FUNCTION FC_CycleTimeToString : STRING(20);
VAR_INPUT
	CycleTime	: DWORD;
END_VAR
VAR
    TempStr : STRING(20);
    Thousands : UDINT;
    Remainder : UDINT;
	sRemainder : STRING(3);
END_VAR

(* Calcolo delle migliaia e del resto *)
Thousands := CycleTime / 1000;
Remainder := CycleTime MOD 1000;

(* Creazione della stringa con il formato richiesto *)
IF Thousands = 0 THEN
    // Se < 1000: stampiamo il valore diretto
	TempStr := '0.';
    TempStr := CONCAT(TempStr, DWORD_TO_STRING(CycleTime));
ELSE
     // Se >= 1000: separiamo migliaia e resto, es. 10901 -> "10.901"
    TempStr := UDINT_TO_STRING(Thousands);

    // Converto il resto in stringa
    sRemainder := UDINT_TO_STRING(Remainder);

    // Aggiungo eventuali zeri a sinistra, per avere sempre 3 cifre nel resto
    IF LEN(sRemainder) = 1 THEN
        sRemainder := CONCAT('00', sRemainder);
    ELSIF LEN(sRemainder) = 2 THEN
        sRemainder := CONCAT('0', sRemainder);
    END_IF

    // Creo la parte "xxx.yyy"
    TempStr := CONCAT(TempStr, '.');
	TempStr := CONCAT(TempStr, sRemainder);
END_IF;

// Aggiungo la " s" finale
FC_CycleTimeToString := CONCAT(TempStr, ' s');

END_FUNCTION

(* stored: Version 1.1.0.1, ProductVersion 3.1.4024.15
   POU FC_CycleTimeToString: Id {32bc795c-1532-4f06-9ce1-df0767ae79d9}, SpecialFunc None *)
